(* IEC 61131-3 sources: InfiniteStateMachine/st/project/infinitestatemachine/function_blocks/statemachine, 5 files *)

(* ---- atlevel-AtLevel.st ---- *)
(* --- Interface --- *)
METHOD PUBLIC AtLevel : IState
VAR_INPUT
	iLevel : INT;
END_VAR

(* --- Implementation --- *)
IF 0 <= iLevel AND iLevel < iDepth THEN
	AtLevel := itfStates[iLevel];
END_IF

(* ---- in-In.st ---- *)
(* --- Interface --- *)
METHOD In : BOOL
VAR_INPUT
	itfState: IState;
END_VAR
VAR
	iLevel : INT := 0;
END_VAR

(* --- Implementation --- *)
(*
 * The following do-while loop's condition assumes early-out semantics.
 * It assumes that the second sub-condition does *not* evaluate unless the first sub-condition is true.
 *)
WHILE iLevel < iDepth AND itfStates[iLevel] <> itfState DO
	iLevel := iLevel + 1;
END_WHILE
In := iLevel < iDepth;

(* ---- leave-Leave.st ---- *)
(* --- Interface --- *)
METHOD PROTECTED Leave
VAR_IN_OUT
	itfState : IState;
END_VAR

(* --- Implementation --- *)
itfState := Pop();
IF itfState <> 0 THEN
	itfState.Leave(THIS^);
END_IF

(* ---- pop-Pop.st ---- *)
(* --- Interface --- *)
METHOD PROTECTED Pop : IState
VAR_INPUT
END_VAR

(* --- Implementation --- *)
IF iDepth > 0 THEN
	iDepth := iDepth - 1;
	Pop := itfStates[iDepth];
    (*
     * Clear the popped state from the stack. This is not strictly necessary,
     * but it can help catch use-after-free bugs.
     *)
	itfStates[iDepth] := 0;
ELSE
	Pop := 0;
END_IF

(* ---- top-Top.st ---- *)
(* --- Interface --- *)
METHOD PUBLIC Top : IState
VAR_INPUT
END_VAR

(* --- Implementation --- *)
IF iDepth > 0 THEN
	Top := itfStates[iDepth - 1];
END_IF
